// TIA Portal V20 export
DATA_BLOCK "CallEquipment_DB"   // DB94
{ DB_Accessible_From_OPC_UA := 'FALSE' }
// stored: AssignedProDiagFB Unit1.Em5.ProDiag, DBAccessibleFromOPCUA false, DBAccessibleFromWebserver false, InstanceOfName Unit1.Em5.CallEquipment, InstanceOfType FB, Namespace Unit1.Em5
"Unit1.Em5.CallEquipment"
   // VAR_INPUT
   //    ZoneOperationEnable { ExternalWritable := 'False'} : "LWONIK_typeSafetyZoneManualOperation";
   //    unitEnableControlInterfaces { ExternalWritable := 'False'} : "LAF_typeEnableControlInterfaces";
   //    commandExcute { ExternalWritable := 'False'} : Bool;
   // END_VAR
   // VAR_IN_OUT
   //    unitStatus : "LAF_typeUnitStatus";
   //    emFeedback : "LUC_typeEmFeedback";
   //    unitAlarmDB : "LAF_typeAlarms";
   // END_VAR
   // VAR
   //    instSequenceManualInput { ExternalWritable := 'False'} : "Unit1.Em5.Sequence_1_ManualInput";
   //    instManualInPutInitializedJob1 { ExternalWritable := 'False'} : "LAF_SelectJob";
   //    instManualInPutLoadingJob2 { ExternalWritable := 'False'} : "LAF_SelectJob";
   //    instManualInPutUnLoaingJob3 { ExternalWritable := 'False'} : "LAF_SelectJob";
   //    instCmNgAndManualInputAxisY { ExternalWritable := 'False'} : "LBC_Axis64Pos_TecPlcCn";
   //    instCmMagazineAxisZ { ExternalWritable := 'False'} : "LBC_Axis64Pos_TecPlcCn";
   //    instCmNgAndManualInputCylinderUpDown { ExternalWritable := 'False'} : "LBC_TwoWayActuatorCn";
   //    instcmNgAndManualInputVacuum1OnOff { ExternalWritable := 'False'} : "LBC_TwoWayActuatorCn";
   //    instCmNgAndManualInputVacuum2OnOff { ExternalWritable := 'False'} : "LBC_TwoWayActuatorCn";
   //    instCmNgAndManualInputVibrator1OnOff { ExternalWritable := 'False'} : "LBC_TwoWayActuatorCn";
   //    instCmNgAndManualInputVibrator2OnOff { ExternalWritable := 'False'} : "LBC_TwoWayActuatorCn";
   //    instcmMagazineLockCylinderUpDown { ExternalWritable := 'False'} : "LBC_TwoWayActuatorCn";
   //    instCmNgAndManaulInputMagazineElectrodeDetectionSensor { ExternalWritable := 'False'} : "LBC_DigitalSignalCn";
   //    instCmNgAndManualInputMagazineDetectionSensor { ExternalWritable := 'False'} : "LBC_DigitalSignalCn";
   //    instCmNgAndManualInputMagazineFullSensor { ExternalWritable := 'False'} : "LBC_DigitalSignalCn";
   //    instCmNgAndManualInputElectrodeDetectionSensor { ExternalWritable := 'False'} : "LBC_DigitalSignalCn";
   //    instcmMagazineSafetyPinIdlePosition { ExternalWritable := 'False'} : "LBC_DigitalSignalCn";
   //    instNgAndManualInputAxisControlInterlockSummary { ExternalWritable := 'False'} : "LER_Axis64Pos_InterlockSummary";
   //    instMagazineAxisControlInterlockSummary { ExternalWritable := 'False'} : "LER_Axis64Pos_InterlockSummary";
   //    instServoTorqueCal_DR7 { ExternalWritable := 'False'} : "LER_ServoTorqueCal";
   //    instServoTorqueCal_DR8 { ExternalWritable := 'False'} : "LER_ServoTorqueCal";
   //    instLDrv701ControlMagazineAxisZ { ExternalWritable := 'False'} : "LDrvSafe_SinaTlg701Control";
   //    instLDrv701StatusMagazineAxisZ { ExternalWritable := 'False'} : "LDrvSafe_SinaTlg701Status";
   //    statUnitStatus { ExternalWritable := 'False'} : "LAF_typeUnitStatus";
   //    statAllBrakeTest { ExternalWritable := 'False'} : "LER_typeBrakeTestUnitCommands";
   //    instManageAlarms { ExternalWritable := 'False'} : "LAF_ManageAlarms";
   //    instEventsPFE { S7_SetPoint := 'True'} : "Unit1.Em5.EventsPFE";
   //    statPulse { ExternalWritable := 'False'} : Array[0..99] of Bool;
   //    statTonTimer { ExternalWritable := 'False'} : Array[0..99] of TON_TIME;
   //    statTofTimer { ExternalWritable := 'False'} : Array[0..99] of TOF_TIME;
   //    statEnableManualCmds { ExternalWritable := 'False'} : Bool;
   //    LoadingCount { ExternalWritable := 'False'} : Int;
   // END_VAR
BEGIN
END_DATA_BLOCK
